FUNCTION_BLOCK FB_CommunicatorClient EXTENDS FB_BaseGroupElement
VAR
END_VAR

METHOD PUBLIC Confirm : BOOL
VAR_INPUT
	sText: STRING;
END_VAR
Confirm		:= THIS^.itfCommunicator.ReceiveDataConfirm (sText := sText, itfRecipient := this^);
END_METHOD

METHOD PUBLIC ReceiveMessage : BOOL
VAR_INPUT
	sText: STRING;
END_VAR

VAR_OUTPUT
	bValue: BOOL;
END_VAR
ReceiveMessage		:= THIS^.itfCommunicator.ReceiveData_BOOL (sText := sText, itfRecipient := THIS^, bValue => bValue);
END_METHOD

METHOD PUBLIC SendMessage : BOOL
VAR_INPUT
	sText: STRING;
END_VAR
SendMessage	:= THIS^.itfCommunicator.SendData_BOOL (sText := sText, itfSender := THIS^);
END_METHOD

END_FUNCTION_BLOCK

(* stored: Version 1.1.0.1, ProductVersion 3.1.4024.15
   POU FB_CommunicatorClient: Id {106a8397-58d1-4356-a1ee-f5b287b3decb}, SpecialFunc None
   Method Confirm: Id {4119d05f-1194-4bdf-ba59-492cedcf1b68}
   Method ReceiveMessage: Id {aedd4f62-5d76-4592-8054-8cb4ea314b46}
   Method SendMessage: Id {67cedbef-3f5f-47d6-88d7-3f00c3c91dff} *)
